TYPE ST_APP_STATE :
STRUCT
  AppInit             : E_PROGRESS;
  State            : E_INSTANCE_STATE;
END_STRUCT
END_TYPE

(* stored: Version 1.1.0.1, ProductVersion 3.1.4026.13
   DUT ST_APP_STATE: Id {2996069c-dabf-495e-beb7-4ffe15dc0c26} *)
